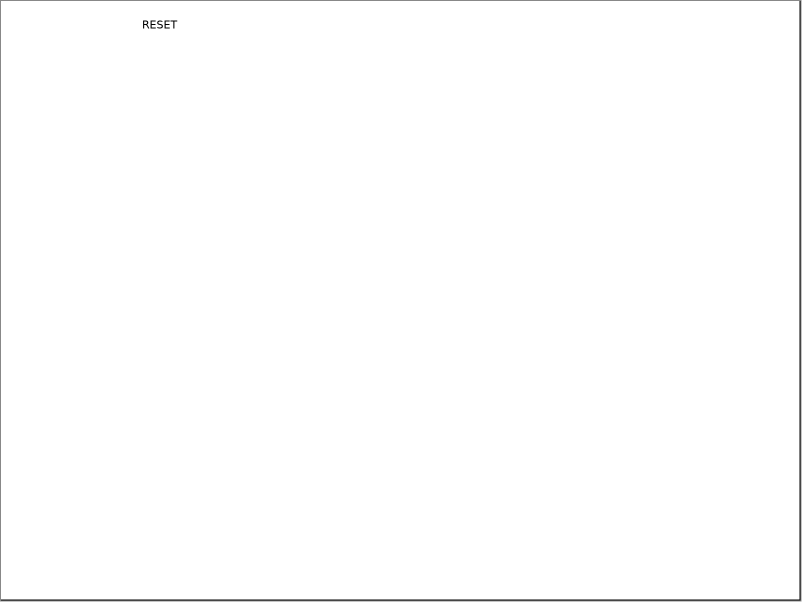
VISUALIZATION F01_Reset  // 802x602
    Rectangle (0,0 800x600)
    Label (10,10 170x30), "RESET"
END_VISUALIZATION

(* stored: Version 1.1.0.1, ProductVersion 3.1.4022.7
   Visu F01_Reset: Id {0ab8e267-e808-48eb-821e-b3a739a15d06} *)
